{attribute 'linkalways'} 
{attribute 'no_explicit_call' := 'This FB is a CLASS and must be accessed using methods or properties'}
{attribute 'enable_dynamic_creation'}
FUNCTION_BLOCK Node_F_VN_FillContainerExp_TcVnPoint3_LREAL EXTENDS VisionNode
VAR
    ipContainer : _ITcVnContainer;
    aValue : _TcVnPoint3_LREAL;
    nStartIdx : _ULINT(0);
    nCount : _ULINT(0);
    hrPrev : _HRESULT(S_OK);
    hresult : _HRESULT(S_OK);
END_VAR

METHOD PUBLIC  Clone : I_Node
VAR
    pNode : POINTER TO Node_F_VN_FillContainerExp_TcVnPoint3_LREAL;
END_VAR
pNode := __NEW(Node_F_VN_FillContainerExp_TcVnPoint3_LREAL);
Clone := pNode^;
END_METHOD

METHOD FB_init : BOOL
VAR_INPUT
    bInitRetains : BOOL; // if TRUE, the retain variables are initialized (warm start / cold start)
    bInCopyCode : BOOL;  // if TRUE, the instance afterwards gets moved into the copy code (online change)
END_VAR
AddInput('ipContainer', ipContainer);
AddInput('aValue', aValue);
AddParameter('nStartIdx', nStartIdx);
AddParameter('nCount', nCount);
AddInput('hrPrev', hrPrev);
AddOutput('ipContainer', ipContainer);
AddOutput('hresult',hresult);
END_METHOD

METHOD PROTECTED OnExecute
hresult.Value := F_VN_FillContainerExp_TcVnPoint3_LREAL(
    ipContainer := ipContainer.Value,
    aValue := aValue.Value,
    nStartIdx := nStartIdx.Value,
    nCount := nCount.Value,
    hrPrev:= hrPrev.Value);
END_METHOD

METHOD PUBLIC PreExecutionCheck
VAR_INPUT
    Check : I_PreExecutionChecks;
END_VAR
Check.IsTrue(ipContainer.IsValid, 'ipContainer must be a valid container');
Check.IsTrue(ipContainer.IsType(TC_GLOBAL_CONST_LIST.ContainerType_Vector_TcVnPoint3_LREAL), 'ipContainer contains incorrect type');
END_METHOD

END_FUNCTION_BLOCK

(* stored: Version 1.1.0.1, ProductVersion 3.1.4026.13
   POU Node_F_VN_FillContainerExp_TcVnPoint3_LREAL: Id {50e4bfc4-abda-4825-84e7-3f649d65f4d5}, SpecialFunc None
   Folder Constructor: Id {d6a8fbbf-52e8-4dfc-b454-6edd40f5c375}
   Method Clone: Id {4d3c999c-c9ea-409f-8a96-44e1dd3787af}
   Method FB_init: Id {42176cc4-ad67-40d9-926d-f67a642d0029}
   Method OnExecute: Id {9b5ebf0e-8bc7-4b14-8b63-7abd491255e3}
   Method PreExecutionCheck: Id {15a9218a-dc15-4e63-a9bb-b55ed86592be} *)
